(* IEC 61131-3 sources: openplc-factoryio-simulator/ladder_logic_project/build, 2 files *)

(* ---- plc.st ---- *)
TYPE
  LOGLEVEL : (CRITICAL, WARNING, INFO, DEBUG) := INFO;
END_TYPE

FUNCTION_BLOCK LOGGER
  VAR_INPUT
    TRIG : BOOL;
    MSG : STRING;
    LEVEL : LOGLEVEL := INFO;
  END_VAR
  VAR
    TRIG0 : BOOL;
  END_VAR

  IF TRIG AND NOT TRIG0 THEN
  {{
   LogMessage(GetFbVar(LEVEL),(char*)GetFbVar(MSG, .body),GetFbVar(MSG, .len));
  }}
  END_IF;
  TRIG0:=TRIG;
END_FUNCTION_BLOCK

PROGRAM ConveyorStarter
  VAR
    visionSensor : BOOL;
    exitSensor : BOOL;
    converyorMotor : BOOL;
  END_VAR

  converyorMotor := NOT(exitSensor) AND visionSensor;
END_PROGRAM

CONFIGURATION Config0

  RESOURCE Res0 ON PLC
    TASK task0(INTERVAL := T#20ms,PRIORITY := 0);
    PROGRAM instance0 WITH task0 : ConveyorStarter;
  END_RESOURCE
END_CONFIGURATION

(* ---- generated_plc.st ---- *)
PROGRAM ConveyorStarter
  VAR
    visionSensor AT %IX0.0 : BOOL;
    exitSensor AT %IX0.2 : BOOL;
    converyorMotor AT %QX0.6 : BOOL;
  END_VAR

  converyorMotor := NOT(exitSensor) AND visionSensor;
END_PROGRAM

CONFIGURATION Config0

  RESOURCE Res0 ON PLC
    TASK task0(INTERVAL := T#20ms,PRIORITY := 0);
    PROGRAM instance0 WITH task0 : ConveyorStarter;
  END_RESOURCE
END_CONFIGURATION
